FUNCTION IsAnyTypeBound : BOOL
VAR_INPUT
	anytype : __SYSTEM.AnyType;
END_VAR

IsAnyTypeBound := anytype.pValue <> 0 AND anytype.diSize > 0;

END_FUNCTION

(* stored: Version 1.1.0.1
   POU IsAnyTypeBound: Id {ef7a7cc5-344a-078b-1ecf-778b92580513}, SpecialFunc None *)
